// TIA Portal V18 export
DATA_BLOCK "MU_Torq_DB"   // DB32
// stored: AutoNumber false, InstanceOfName MU_Torq, InstanceOfType FB
"MU_Torq"
   // VAR_INPUT
   //    Start : Bool;
   // END_VAR
   // VAR_OUTPUT
   //    FlowFwdmAOut : Real;
   //    TorqmAOut : Real;
   //    EnableP1 : Bool;
   //    EnableP2 { ExternalWritable := 'False'} : Bool;
   //    TorqEn : Bool;
   //    MUSeqRunning : Bool;
   // END_VAR
   // VAR
   //    MUspeed : Real;
   //    PumpToggle : Bool;
   //    AutoMUComplete : Bool;
   //    RampDown : Bool;
   //    RampDownComplete : Bool;
   //    MUComplete_TON { S7_SetPoint := 'True'} : TON_TIME;
   //    TorqUserSetmA : Real;
   //    AutoMUInc_TON { S7_SetPoint := 'True'} : TON_TIME;
   //    Torq_Ramp { S7_SetPoint := 'True'} : RampFunction;
   //    Flow_Ramp { S7_SetPoint := 'True'} : RampFunction;
   //    TorqRampInmA { S7_SetPoint := 'True'} : Real;
   //    FlowRampInmA : Real;
   //    MUSeqRunLast : Bool;
   // END_VAR
BEGIN
END_DATA_BLOCK
